INTERFACE I_DefaultHomingBuilder EXTENDS __System.IQueryInterface

METHOD BuildDefaultHomingCommand : I_HomingCommand
END_METHOD

METHOD Cam : I_DefaultHomingBuilder
VAR_INPUT
	value : REFERENCE TO BOOL;
END_VAR
END_METHOD

METHOD ClearLag : I_PositioningHomingBuilder
END_METHOD

METHOD KeepLag : I_PositioningHomingBuilder
END_METHOD

METHOD Position : I_PositioningHomingBuilder
VAR_INPUT
	value : LREAL;
END_VAR
END_METHOD

METHOD ReferenceMode : I_DefaultHomingBuilder
VAR_INPUT
	value : EncoderReferenceMode;
END_VAR
END_METHOD

METHOD SearchDirection : I_DefaultHomingBuilder
VAR_INPUT
	value : Direction;
END_VAR
END_METHOD

METHOD SearchVelocity : I_DefaultHomingBuilder
VAR_INPUT
	value : LREAL;
END_VAR
END_METHOD

METHOD SyncDirection : I_DefaultHomingBuilder
VAR_INPUT
	value : Direction;
END_VAR
END_METHOD

METHOD SyncVelocity : I_DefaultHomingBuilder
VAR_INPUT
	value : LREAL;
END_VAR
END_METHOD

END_INTERFACE

(* stored: Version 1.1.0.1, ProductVersion 3.1.4024.12
   Itf I_DefaultHomingBuilder: Id {5ea10c40-2902-4ebb-9cb2-4e71ecc68835}
   Method BuildDefaultHomingCommand: Id {3dc16efd-5cb8-45e4-8d34-7cce92aaad75}
   Method Cam: Id {c1d8e263-3982-4713-948b-cc0ec7a108ac}
   Method ClearLag: Id {d3c63066-cd1a-48b8-9819-bf97ba0ad83e}
   Method KeepLag: Id {d473dabf-8ee5-4466-b736-393d1842fb4b}
   Method Position: Id {85eefe23-3d7c-493a-a578-54830cc3878b}
   Method ReferenceMode: Id {2b594bd4-7168-4ca5-8d51-5740d31c94ba}
   Method SearchDirection: Id {f65bac35-534a-4861-b4b4-02efc84a84b8}
   Method SearchVelocity: Id {8e5e7dd0-6ef6-413e-a368-3487e41d4b51}
   Method SyncDirection: Id {14b7130d-d9df-4207-bd4f-34c428bfaf5b}
   Method SyncVelocity: Id {e4f7a142-d8a7-4720-8b79-8be80462907c} *)
